Staubli VAL3: refresh.pgx

program refresh()
// // page refresh
begin
  if !use:bShowDialog and !cycleStatus:bShowMessage
    //
    // refresh the static message
    if (nKey>=270 and nKey<=278) or (nKey==264 or nKey==268) or (use:bUseRefresh and !bShowStatus)
      call refreshStatic()
      call refreshDynamic()
    else
      if !bShowStatus
        // refresh the Dynamic message
        if abs(clock()-nRefresh)>nTime
          call refreshDynamic()
        endIf
      endIf
    endIf
  endIf
  //
  call showStatus()
end
